Yaskawa INFORM job: SKRZYNIA_5340_0_STOPNI_1OBR.JBI

/JOB
//NAME SKRZYNIA_5340_0_STOPNI_1OBR
///FOLDERNAME 02-SKRZYNIE_JOBS
//POS
///NPOS 610,610,0,47,4,0
///TOOL 0
///POSTYPE PULSE
///PULSE
C00000=1055,-24125,84372,288,19725,204
C00001=1055,-24125,84372,288,19725,204
C00002=0,-15438,65714,0,-68532,0
C00003=25524,-25821,36823,19654,-58495,38520
C00004=23988,-24960,37134,18595,-57837,38812
C00005=22822,-23954,37534,17811,-57199,39017
C00006=22935,-24057,37491,17887,-57262,38997
C00007=20006,-24258,37408,15644,-56932,39751
C00008=24402,-25289,37013,18874,-58060,38740
C00009=22585,-24665,40358,17164,-59622,30036
C00010=23477,-23257,40205,18030,-58646,29630
C00011=22519,-22398,40568,17384,-58125,29795
C00012=22700,-22567,40495,17506,-58225,29764
C00013=19339,-22794,40398,14955,-57865,30607
C00014=24825,-24328,39798,18931,-59350,29401
C00015=32755,-32613,25711,29640,-48730,33694
C00016=25632,-30899,26166,23992,-46203,35378
C00017=24264,-29862,26497,22996,-45413,35639
C00018=24403,-29974,26459,23097,-45496,35612
C00019=20575,-30233,26374,19602,-44891,36810
C00020=26556,-31526,25988,24663,-46720,35206
C00021=30846,-32795,25752,28021,-48338,30427
C00022=24953,-30697,26306,23444,-45946,31743
C00023=23937,-29910,26558,22702,-45353,31936
C00024=24039,-29993,26530,22778,-45414,31916
C00025=20322,-30240,26449,19379,-44834,33080
C00026=25997,-31433,26093,24205,-46535,31545
C00027=26028,-43665,26580,-39946,8682,24640
C00028=27956,-30595,53065,-101898,6609,54413
C00029=26028,-43663,26580,-39944,8677,24639
C00030=38784,-34544,25404,33956,-51320,34445
C00031=29266,-32676,25756,26732,-47889,36488
C00032=25734,-31262,26119,24020,-46377,37252
C00033=24289,-30200,26441,22967,-45549,37525
C00034=24367,-30262,26420,23025,-45594,37511
C00035=20043,-30544,26331,19080,-44922,38860
C00036=26573,-31816,25967,24631,-46839,37095
C00037=27817,-32566,25782,25532,-47502,36865
C00038=25779,-31294,26110,24054,-46400,37243
C00039=24344,-30243,26427,23007,-45578,37515
C00040=24432,-30312,26405,23072,-45630,37498
C00041=20021,-30599,26315,19050,-44944,38872
C00042=26262,-31616,26021,24405,-46667,37153
C00043=27439,-32346,25835,25259,-47302,36935
C00044=25570,-31108,26163,23910,-46262,37277
C00045=24581,-30384,26384,23190,-45695,37464
C00046=24689,-30466,26358,23269,-45758,37444
C00047=20001,-30771,26264,18999,-45026,38899
C00048=26308,-31607,26026,24448,-46671,37139
C00049=27526,-32360,25834,25329,-47326,36914
C00050=24269,-40076,6479,29767,-34177,34232
C00051=22958,-37632,10123,27061,-35370,35326
C00052=22703,-41294,1722,31272,-29953,33282
C00053=19440,-41515,1663,27208,-29122,34832
C00054=25465,-43501,1200,33269,-31905,32752
C00055=87177,-39066,-1236,81808,-72661,19198
C00056=4794,-34097,38974,4189,-31824,-1302
C00057=4794,-34097,38974,4189,13412,-1302
C00058=11237,-37131,38982,-12694,5333,8253
C00059=6591,-33902,35532,5956,-1761,-1932
C00060=10065,-33530,28876,9373,-31104,-3154
C00061=31877,-32319,25770,29025,-48287,33360
C00062=24706,-30765,26196,23236,-45867,35119
C00063=23652,-29939,26460,22464,-45250,35320
C00064=23742,-30013,26436,22530,-45305,35302
C00065=19630,-30281,26348,18756,-44677,36597
C00066=26056,-31710,25928,24219,-46631,34863
C00067=38095,-40136,7813,41252,-44156,24924
C00068=33231,-38681,8176,37792,-41757,25918
C00069=31538,-37640,8473,36716,-40716,26179
C00070=31687,-37737,8444,36811,-40809,26155
C00071=27389,-38154,8322,32773,-39589,27627
C00072=33834,-39023,8084,38175,-42120,25821
C00073=27585,-47842,-289,32095,-40789,28095
C00074=4801,-35772,25187,4593,-28023,-82032
C00075=17634,-23800,39238,9573,-31425,-73339
C00076=17634,-23800,39238,9573,-31425,-73339
C00077=16549,-22464,39800,8390,-30730,-72975
C00078=16684,-22641,39722,8536,-30818,-73021
C00079=16684,-19968,45512,8078,-32771,-72767
C00080=17634,-23800,39238,9573,-31425,-73339
C00081=17837,-21535,44509,9322,-33342,-73155
C00082=17837,-21535,44509,9322,-33342,-73155
C00083=16866,-20378,45014,8305,-32755,-72853
C00084=17032,-20588,44918,8481,-32857,-72905
C00085=17032,-17542,51480,8009,-35060,-72636
C00086=17837,-21535,44509,9322,-33342,-73155
C00087=-20829,-18800,50532,-12466,-37179,-77446
C00088=-19934,-17904,50946,-11618,-36715,-77676
C00089=-20044,-18019,50891,-11723,-36773,-77647
C00090=-20044,-15288,56753,-11218,-38713,-77950
C00091=-20966,-18928,50473,-12596,-37250,-77413
C00092=-20884,-26676,33664,-14451,-31668,-76336
C00093=-20884,-26676,33664,-14451,-31668,-76336
C00094=-19557,-25338,34176,-13080,-30873,-76751
C00095=-19691,-25483,34117,-13220,-30955,-76709
C00096=-19691,-22773,39998,-12506,-32911,-77106
C00097=-20642,-26447,33747,-14206,-31526,-76411
C00098=-33629,-40566,17444,-29603,-33447,-71192
C00099=-33629,-40566,17444,42578,-32312,-84654
C00100=-42160,-31266,16400,42578,-32312,-84654
C00101=-87798,-804,48829,-20188,-26072,-60966
C00102=-76454,-11934,10236,-25964,7954,-64922
C00103=-76448,-11928,10235,-25961,7944,-64914
C00104=-68643,-7759,-23318,-14097,50582,-74897
C00105=-70868,-8793,-8075,-29663,30364,-70765
C00106=-67243,-1968,12282,-49553,26687,-63567
C00107=-68655,-309,14069,-48513,25966,-64203
C00108=-67497,-1678,12591,-49367,26558,-63682
C00109=-71436,-723,2905,-26484,35140,-73726
C00110=-71436,176,6426,-27636,33595,-73066
C00111=-71434,778,8668,-28412,32633,-72624
C00112=-68624,-2689,-85,-28291,36551,-72622
C00113=-99375,3692,5712,40719,48607,-84097
C00114=-94964,4957,10918,40408,44640,-83792
C00115=-93063,6047,12199,39572,43744,-83178
C00116=-94964,4957,10918,40408,44640,-83792
C00117=-94964,5754,13918,41385,43553,-84439
C00118=-94964,4957,10918,40408,44640,-83792
C00119=-90271,-412,-5146,23417,46876,-76529
C00120=-83133,-4088,-8267,6704,41492,-71542
C00121=-83133,-4088,-8267,6704,41492,-71542
C00122=-83133,-4088,-8267,6704,41492,-11598
C00123=-83133,-16026,-8267,6704,41492,-11598
C00124=-83133,-16026,-8267,6704,41492,-11598
C00125=-48225,-19387,30619,3889,32460,-6728
C00126=56943,-39861,25115,1795,-37402,-69601
C00127=29960,-38386,-19607,-115769,-41858,-24264
C00128=65721,-6478,18155,-133323,-22195,3361
C00129=70544,4411,32968,-134868,-18623,4660
C00130=71874,8263,38598,-134556,-17327,4659
C00131=72629,9390,40002,-135279,-16924,5107
C00132=71441,7638,37831,-134139,-17555,4406
C00133=77146,8888,25050,-166574,-32612,18372
C00134=77146,10029,28643,-166204,-31014,18167
C00135=77146,11198,32202,-165803,-29459,17947
C00136=75508,4678,16951,-165715,-35157,17778
C00137=68680,12216,24468,-164340,-40455,-13359
C00138=68362,12845,25743,-164045,-40097,-13561
C00139=68362,13700,28585,-163752,-38808,-13742
C00140=68362,12845,25743,-164045,-40097,-13561
C00141=64993,-1168,28876,-102971,-10760,-49875
C00142=63888,481,30670,-102324,-11438,-50313
C00143=64993,-1168,28876,-102971,-10760,-49875
C00144=4264,-34194,25387,4006,-26954,-29436
C00145=4264,-34194,25387,4006,-26954,-81856
C00146=17634,-23800,39238,9573,-31425,-73339
C00147=17837,-27228,32238,10495,-29236,-73805
C00148=17837,-21535,44509,9322,-33342,-73155
C00149=17548,-20734,45666,8935,-33511,-73021
C00150=-20829,-18800,50532,-12466,-37179,-77446
C00151=-20884,-20901,46110,-12960,-35762,-77182
C00152=-20884,-26676,33664,-14451,-31668,-76336
C00153=-20624,-26699,33167,-14265,-31320,-76369
C00154=-33629,-40566,17444,-29603,-33447,-71192
C00155=-33629,-40566,17444,42578,-32312,-84654
C00156=-42160,-31266,16400,42578,-32312,-84654
C00157=-87798,-804,48829,-20188,-26072,-60966
C00158=-76454,-11934,10236,-25964,7954,-64922
C00159=-76448,-11928,10235,-25961,7944,-64914
C00160=-68643,-7759,-23318,-14097,50582,-74897
C00161=-70868,-8793,-8075,-29663,30364,-70765
C00162=-67243,-1968,12282,-49553,26687,-63567
C00163=-68655,-309,14069,-48513,25966,-64203
C00164=-67497,-1678,12591,-49367,26558,-63682
C00165=-71436,-723,2905,-26484,35140,-73726
C00166=-71436,176,6426,-27636,33595,-73066
C00167=-71434,778,8668,-28412,32633,-72624
C00168=-68624,-2689,-85,-28291,36551,-72622
C00169=-99375,3692,5712,40719,48607,-84097
C00170=-94964,4957,10918,40408,44640,-83792
C00171=-93063,6047,12199,39572,43744,-83178
C00172=-94964,4957,10918,40408,44640,-83792
C00173=-94964,5754,13918,41385,43553,-84439
C00174=-94964,4957,10918,40408,44640,-83792
C00175=-90271,-412,-5146,23417,46876,-76529
C00176=-83133,-4088,-8267,6704,41492,-71542
C00177=-83133,-4088,-8267,6704,41492,-71542
C00178=-83133,-4088,-8267,6704,41492,-11598
C00179=-83133,-16026,-8267,6704,41492,-11598
C00180=-83133,-16026,-8267,6704,41492,-11598
C00181=-48225,-19387,30619,3889,32460,-6728
C00182=56943,-39861,25115,1795,-37402,-69601
C00183=29960,-38386,-19607,-115769,-41858,-24264
C00184=65721,-6478,18155,-133323,-22195,3361
C00185=70544,4411,32968,-134868,-18623,4660
C00186=71874,8263,38598,-134556,-17327,4659
C00187=72629,9390,40002,-135279,-16924,5107
C00188=71441,7638,37831,-134139,-17555,4406
C00189=77146,8888,25050,-166574,-32612,18372
C00190=77146,10029,28643,-166204,-31014,18167
C00191=77146,11198,32202,-165803,-29459,17947
C00192=75508,4678,16951,-165715,-35157,17778
C00193=68680,12216,24468,-164340,-40455,-13359
C00194=68362,12845,25743,-164045,-40097,-13561
C00195=68362,13700,28585,-163752,-38808,-13742
C00196=68362,12845,25743,-164045,-40097,-13561
C00197=64993,-1168,28876,-102971,-10760,-49875
C00198=63888,481,30670,-102324,-11438,-50313
C00199=64993,-1168,28876,-102971,-10760,-49875
C00200=58588,-14653,4620,-120782,-19611,-35794
C00201=29960,-38386,-19607,-115769,-41858,-24264
C00202=56943,-39861,25115,1795,-37402,-69601
C00203=-1002,-39861,25115,1795,-37402,-69601
C00204=-1001,-39858,25114,1795,-37402,0
C00205=6591,-33902,35532,5956,-1761,-1932
C00206=6592,-33900,35531,103508,-35512,-26314
C00207=-99253,-13690,44082,59847,13407,-31313
C00208=-85045,-36869,-4353,28502,-22832,-52282
C00209=-92346,-18713,13565,21110,-22545,-55257
C00210=-85370,-14218,16934,32905,-23649,-60330
C00211=-84150,-13282,17685,34842,-23935,-61163
C00212=-82877,-12536,18624,36445,-24482,-61818
C00213=-84150,-13282,17685,34842,-23935,-61163
C00214=-85467,-11480,19558,33086,-23405,-60436
C00215=-84150,-13282,17685,34842,-23935,-61163
C00216=-85732,-21202,11427,30682,-24763,-59235
C00217=-84559,-15616,15722,33768,-24118,-60665
C00218=-84150,-13282,17685,34842,-23935,-61163
C00219=-83260,-12880,18034,36130,-24218,-61709
C00220=-84150,-13282,17685,34842,-23935,-61163
C00221=-85365,-11775,19006,33430,-23307,-60600
C00222=-84150,-13282,17685,34842,-23935,-61163
C00223=-85786,-16909,14677,31743,-23900,-59790
C00224=-84150,-13282,17685,34842,-23935,-61163
C00225=-83215,-12861,18051,36194,-24233,-61735
C00226=-84150,-13282,17685,34842,-23935,-61163
C00227=-85327,-11825,18959,33476,-23327,-60618
C00228=-84150,-13282,17685,34842,-23935,-61163
C00229=-87841,-18519,13420,28367,-23534,-58339
C00230=-84150,-13282,17685,34842,-23935,-61163
C00231=-83292,-12894,18020,36083,-24208,-61688
C00232=-84150,-13282,17685,34842,-23935,-61163
C00233=-85185,-12008,18799,33646,-23400,-60687
C00234=-84150,-13282,17685,34842,-23935,-61163
C00235=-86371,-18277,13606,30568,-23951,-59265
C00236=-84345,-13370,17612,34554,-23873,-61041
C00237=-83240,-12871,18042,36158,-24225,-61720
C00238=-84345,-13370,17612,34554,-23873,-61041
C00239=-85365,-12110,18711,33368,-23345,-60568
C00240=-84345,-13370,17612,34554,-23873,-61041
C00241=-86191,-19647,12567,30467,-24278,-59187
C00242=-84345,-13372,17610,34552,-23873,-61039
C00243=-83096,-12807,18098,36363,-24268,-61804
C00244=-84345,-13372,17610,34552,-23873,-61039
C00245=-85268,-12232,18600,33480,-23393,-60612
C00246=-84345,-13372,17610,34552,-23873,-61039
C00247=-84814,-16043,15376,33312,-24093,-60464
C00248=-84104,-13265,17702,34906,-23948,-61189
C00249=-82960,-12743,18153,36555,-24313,-61887
C00250=-84104,-13265,17702,34906,-23948,-61189
C00251=-84979,-12194,18635,33901,-23496,-60788
C00252=-84104,-13265,17702,34906,-23948,-61189
C00253=-86610,-16845,14732,30573,-23614,-59301
C00254=-84104,-13265,17702,34906,-23948,-61189
C00255=-82793,-12667,18222,36790,-24370,-61986
C00256=-84104,-13265,17702,34906,-23948,-61189
C00257=-84888,-12305,18537,34004,-23540,-60830
C00258=-84104,-13265,17702,34906,-23948,-61189
C00259=-83806,-19585,12613,33764,-25080,-60559
C00260=-83675,-13072,17868,35530,-24083,-61453
C00261=-82553,-12556,18319,37130,-24451,-62127
C00262=-83675,-13072,17868,35530,-24083,-61453
C00263=-84378,-12223,18610,34735,-23716,-61138
C00264=-83675,-13072,17868,35530,-24083,-61453
C00265=-87149,-17993,13826,29513,-23647,-58830
C00266=-84104,-13265,17702,34906,-23948,-61189
C00267=-82640,-12594,18285,37014,-24425,-62079
C00268=-84104,-13265,17702,34906,-23948,-61189
C00269=-84792,-12429,18430,34119,-23592,-60877
C00270=-84104,-13265,17702,34906,-23948,-61189
C00271=-83583,-9185,30892,23668,-36042,-57025
C00272=-85789,-8328,35795,20592,-37093,-55378
C00273=-85786,-16735,14816,31782,-23869,-59812
C00274=-84103,-13263,17702,34906,-23947,-61191
C00275=-83225,-12865,18046,36177,-24227,-61729
C00276=-84103,-13263,17702,34906,-23947,-61191
C00277=-84774,-12447,18412,34138,-23599,-60886
C00278=-84103,-13263,17702,34906,-23947,-61191
C00279=-86149,-16246,6730,18897,-35239,-57128
C00280=-86244,-15289,7532,18875,-35060,-57127
C00281=-85361,-14893,7870,19824,-35193,-57574
C00282=-86244,-15289,7532,18875,-35060,-57127
C00283=-86889,-14409,8282,18264,-34784,-56850
C00284=-86244,-15289,7532,18875,-35060,-57127
C00285=-90262,-21765,2389,14114,-35574,-54847
C00286=-90262,-21765,2389,28730,-17672,-54847
C00287=-89967,-19086,25635,28730,-17672,-54847
C00288=568,-24029,84339,168,19981,112
C00289=568,-24677,83015,164,20405,113
C00290=101153,-24598,83176,165,20353,113
C00291=101153,-24598,83176,165,20353,113
C00292=89967,-19086,25635,-28730,-17672,54847
C00293=90262,-21765,2389,-28730,-17672,54847
C00294=86932,-18662,4771,-17876,-35519,56628
C00295=86578,-15436,7408,-18515,-35011,56957
C00296=85428,-14922,7844,-19753,-35183,57541
C00297=84405,-14447,8250,-20842,-35348,58054
C00298=85428,-14922,7844,-19753,-35183,57541
C00299=86134,-13973,8661,-19091,-34881,57237
C00300=85428,-14922,7844,-19753,-35183,57541
C00301=85786,-16735,14816,-31782,-23869,59812
C00302=83514,-12996,17929,-35760,-24132,61552
C00303=82296,-12429,18424,-37488,-24534,62281
C00304=83514,-12996,17929,-35760,-24132,61552
C00305=84266,-12085,18725,-34910,-23738,61214
C00306=83514,-12996,17929,-35760,-24132,61552
C00307=87323,-6914,39851,-18853,-38149,44508
C00308=83118,-12818,18089,-36330,-24263,61791
C00309=81969,-12276,18566,-37944,-24648,62472
C00310=83118,-12818,18089,-36330,-24263,61791
C00311=83927,-11846,18941,-35423,-23842,61433
C00312=83118,-12818,18089,-36330,-24263,61791
C00313=83806,-19585,12613,-33764,-25080,60559
C00314=83148,-12832,18077,-36287,-24254,61773
C00315=81889,-12236,18598,-38058,-24676,62520
C00316=83148,-12832,18077,-36287,-24254,61773
C00317=83900,-11930,18867,-35446,-23862,61440
C00318=83148,-12832,18077,-36287,-24254,61773
C00319=86610,-16845,14732,-30573,-23614,59301
C00320=82493,-13239,17725,-37070,-24559,62089
C00321=81442,-12739,18159,-38529,-24915,62703
C00322=82493,-13239,17725,-37070,-24559,62089
C00323=83435,-12133,18689,-36040,-24063,61682
C00324=82493,-13239,17725,-37070,-24559,62089
C00325=84814,-16043,15376,-33312,-24093,60464
C00326=82555,-13613,17404,-36910,-24580,62015
C00327=81369,-13053,17885,-38558,-24979,62709
C00328=82555,-13613,17404,-36910,-24580,62015
C00329=83568,-12431,18429,-35805,-24046,61580
C00330=82555,-13613,17404,-36910,-24580,62015
C00331=86191,-19647,12567,-30467,-24278,59187
C00332=82500,-13648,17375,-36975,-24607,62039
C00333=81594,-13224,17740,-38236,-24911,62571
C00334=82500,-13648,17375,-36975,-24607,62039
C00335=83449,-12543,18332,-35941,-24104,61633
C00336=82500,-13648,17375,-36975,-24607,62039
C00337=86371,-18277,13606,-30568,-23951,59265
C00338=82904,-13790,17251,-36416,-24470,61808
C00339=81796,-13275,17692,-37971,-24838,62464
C00340=82904,-13790,17251,-36416,-24470,61808
C00341=83696,-12867,18046,-35547,-24051,61466
C00342=82904,-13790,17251,-36416,-24470,61808
C00343=87841,-18519,13420,-28367,-23534,58339
C00344=82748,-13879,17174,-36603,-24542,61883
C00345=81789,-13434,17554,-37946,-24861,62449
C00346=82748,-13879,17174,-36603,-24542,61883
C00347=83603,-12888,18026,-35668,-24086,61514
C00348=82748,-13879,17174,-36603,-24542,61883
C00349=85786,-16909,14677,-31743,-23900,59790
C00350=82339,-14116,16972,-37087,-24733,62079
C00351=81557,-13752,17280,-38171,-24994,62536
C00352=82339,-14116,16972,-37087,-24733,62079
C00353=83390,-12909,18006,-35951,-24172,61633
C00354=82339,-14116,16972,-37087,-24733,62079
C00355=85732,-21202,11427,-30682,-24763,59235
C00356=82398,-14365,16763,-36952,-24745,62014
C00357=81340,-13876,17176,-38416,-25096,62632
C00358=82398,-14365,16763,-36952,-24745,62014
C00359=83629,-12951,17972,-35620,-24090,61491
C00360=82398,-14365,16763,-36952,-24745,62014
C00361=92346,-18713,13565,-21110,-22545,55257
C00362=82794,-13980,17083,-36511,-24538,61844
C00363=81697,-13472,17516,-38043,-24902,62488
C00364=82794,-13980,17083,-36511,-24538,61844
C00365=83767,-12847,18056,-35444,-24023,61424
C00366=82794,-13980,17083,-36511,-24538,61844
C00367=85045,-36869,-4353,-28502,-22832,52282
C00368=69856,-53931,-13446,-33557,-28911,29591
C00369=73943,-28815,39553,-16801,-45089,19004
C00370=0,-24029,84339,0,19981,0
C00371=0,-24029,84339,0,19981,0
C00372=0,-52280,40443,0,6876,0
C00373=63961,-36661,14391,66570,-58199,13439
C00374=50233,-31965,16595,55443,-54435,15843
C00375=47147,-32819,12541,55607,-51124,17230
C00376=46896,-37872,871,62973,-46008,11193
C00377=54160,-39955,137,66075,-50361,10746
C00378=0,-52280,40443,0,6876,0
C00379=0,-52280,40443,1,6876,0
C00380=42978,-45587,7631,48214,-41849,18034
C00381=34615,-32719,24207,35617,-45539,22507
C00382=46734,-24688,30880,50025,-55713,21863
C00383=45059,-39151,-3508,69830,-41334,11649
C00384=32474,-45233,-13338,65386,-28486,22104
C00385=59828,-44646,-5405,72855,-48572,12139
C00386=0,-38761,66314,0,-763,0
C00387=0,-44757,54667,0,2744,0
C00388=40382,-38226,12225,48505,-40693,16039
C00389=55481,-27484,23768,62968,-54833,11978
C00390=49931,-26522,24223,59987,-51967,12537
C00391=49591,-31309,12277,55066,-55958,13102
C00392=55330,-33748,11238,57660,-59334,12681
C00393=78664,-24436,10378,82837,-79111,12029
C00394=75189,-23065,11287,81851,-76948,11927
C00395=75189,-45249,11287,81851,-38847,11927
C00396=29880,-45249,11287,43145,-11324,11927
C00397=0,-24029,84339,0,19981,0
C00398=0,-24026,84338,1,19977,2
C00399=4264,-34194,25387,4006,-26954,-29436
C00400=4264,-34194,25387,4006,-26954,-81856
C00401=-21478,-27798,32214,-15234,-31599,-76056
C00402=-19679,-23059,39354,-12567,-32689,-77067
C00403=16724,-20576,44291,8212,-32395,-72836
C00404=21329,-26386,39716,13285,-34016,-74401
C00405=-23778,-26243,38799,-16502,-35132,-75964
C00406=-20075,-15782,55752,-11329,-38404,-77896
C00407=16874,-17447,51356,7863,-34895,-72604
C00408=18580,-28601,30698,11472,-29284,-74138
C00409=6126,-41331,18955,6697,-26557,-30383
C00410=1,-24024,84337,2,19973,1
C00411=-64243,-26178,31107,-39513,40312,-5844
C00412=-72148,3973,56008,-35470,42045,-10522
C00413=-72090,16396,76301,-42067,35650,-6519
C00414=-69388,15725,61378,-31740,35177,-8719
C00415=-69127,27099,75569,-32744,34250,-8088
C00416=-67573,2495,11285,-21767,57629,-15193
C00417=-77819,19629,29798,-10454,63174,-20704
C00418=-72990,23583,14304,-10735,77209,-20379
C00419=-74593,38003,46707,-11043,65751,-19814
C00420=-73236,38943,48295,-11400,65557,-19316
C00421=-73329,42107,51779,-6346,67443,-19636
C00422=-87142,34654,46174,17622,63862,-25393
C00423=-87240,36727,48611,18897,66604,-25032
C00424=-99033,21517,12213,24947,79702,-26203
C00425=-91500,-14196,-34781,24472,81625,-22832
C00426=-100472,-45007,-27818,8167,67201,-29302
C00427=0,-36642,16905,0,48372,0
C00428=66009,-61997,-62105,21406,63483,18379
C00429=97242,-23579,-39442,10179,68876,30321
C00430=73684,-7073,-17511,24638,68131,29022
C00431=59136,7235,6676,33270,66602,27507
C00432=54816,14937,6234,39741,69494,31070
C00433=54365,20668,19279,41017,66202,29418
C00434=64503,4223,2857,29650,48528,26647
C00435=75622,3202,-3149,3890,49494,34281
C00436=88036,13177,2413,-18568,66573,35876
C00437=90462,21593,10123,-22613,76266,34479
C00438=92450,29224,20002,-25750,81642,33727
C00439=94949,8131,-12163,-20291,74229,36861
C00440=94949,8084,-13484,-20215,75047,36712
C00441=70412,-34016,-52305,-11724,65624,29757
C00442=18580,-28601,30698,11472,-29284,-74138
C00443=-23778,-26243,38799,-16502,-35132,-75964
C00444=18580,-28601,30698,11472,-29284,-74138
C00445=4264,-34194,25387,4006,-26954,-81856
C00446=4264,-34194,25387,4006,-26954,-29436
C00447=1,-24024,84337,2,19973,1
C00448=-64243,-26178,31107,-39513,40312,-5844
C00449=-72148,3973,56008,-35470,42045,-10522
C00450=-72090,16396,76301,-42067,35650,-6519
C00451=-69388,15725,61378,-31740,35177,-8719
C00452=-69127,27099,75569,-32744,34250,-8088
C00453=-67573,2495,11285,-21767,57629,-15193
C00454=-77819,19629,29798,-10454,63174,-20704
C00455=-72990,23583,14304,-10735,77209,-20379
C00456=-74593,38003,46707,-11043,65751,-19814
C00457=-73236,38943,48295,-11400,65557,-19316
C00458=-73329,42107,51779,-6346,67443,-19636
C00459=-87142,34654,46174,17622,63862,-25393
C00460=-87240,36727,48611,18897,66604,-25032
C00461=-99033,21517,12213,24947,79702,-26203
C00462=-91500,-14196,-34781,24472,81625,-22832
C00463=-100472,-45007,-27818,8167,67201,-29302
C00464=0,-36642,16905,0,48372,0
C00465=66009,-61997,-62105,21406,63483,18379
C00466=97242,-23579,-39442,10179,68876,30321
C00467=73684,-7073,-17511,24638,68131,29022
C00468=59136,7235,6676,33270,66602,27507
C00469=54816,14937,6234,39741,69494,31070
C00470=54365,20668,19279,41017,66202,29418
C00471=64503,4223,2857,29650,48528,26647
C00472=75622,3202,-3149,3890,49494,34281
C00473=88036,13177,2413,-18568,66573,35876
C00474=90462,21593,10123,-22613,76266,34479
C00475=92450,29224,20002,-25750,81642,33727
C00476=94949,8131,-12163,-20291,74229,36861
C00477=94949,8084,-13484,-20215,75047,36712
C00478=70412,-34016,-52305,-11724,65624,29757
C00479=44268,-30306,-1568,-7370,48673,18708
C00480=1,-24024,84337,2,19973,1
C00481=1,-24024,84337,2,19973,1
C00482=3796,-57671,22373,2336,-25309,-753
C00483=52632,-34554,16626,51161,-63050,5622
C00484=59461,-32779,9832,66317,-58406,17312
C00485=52745,-27759,19165,60340,-56543,14824
C00486=51596,-17381,41670,51728,-64721,19335
C00487=62932,-33588,12189,66848,-61063,18031
C00488=1,-24024,84337,2,19973,1
C00489=1,-24024,84337,2,19973,1
C00490=57188,-41777,19973,48132,-58706,4905
C00491=55566,-48748,-16991,79805,-45048,-6941
C00492=49908,-48716,-25784,90749,-41340,-3650
C00493=44060,-47282,-25482,90760,-37623,-4446
C00494=43373,-46910,-25348,90885,-37191,-4606
C00495=55479,-50244,-26473,91085,-44870,-3042
C00496=12119,-24859,71505,13236,4440,2633
C00497=-91085,-34291,10385,1908,-24348,-42097
C00498=-86191,-19647,12567,30467,-24278,-59187
C00499=-99148,-11667,19101,-13975,-20192,-40187
C00500=-98206,-11518,19604,-10142,-20308,-41629
C00501=-99474,-20389,12397,-11593,-22150,-41069
C00502=0,-52280,40443,0,6876,0
C00503=85348,-24204,23536,-13963,-15515,44275
C00504=84670,-17015,14597,-33277,-24304,60423
C00505=96971,-12584,18294,8365,-19955,42614
C00506=97182,-12918,18001,8747,-20027,42449
C00507=96230,-24528,9149,6144,-22576,43630
C00508=0,-52280,40443,0,6876,0
C00509=0,-52280,40443,0,6876,0
C00510=-90140,-60305,18108,-2708,1721,-7625
C00511=-95594,-27428,6866,-4663,-19832,-42154
C00512=-99356,-13410,18355,-15385,-17730,-37479
C00513=-99405,-10878,20508,-15853,-17333,-37255
C00514=-99132,-10804,20575,-15274,-17279,-37502
C00515=-99132,-3482,39129,-10940,-24351,-39674
C00516=-98851,-3328,38974,-10588,-24101,-39807
C00517=-100183,-18601,14070,-16273,-18800,-37146
C00518=-90140,-60305,18108,-2708,1721,-7625
C00519=0,-52280,40443,0,6876,0
C00520=84259,-57935,27522,-3761,3673,6310
C00521=86507,-39672,4297,-27618,-16640,46340
C00522=70477,-27878,7073,-45786,-32339,64941
C00523=84043,-16293,15174,-34312,-24409,60872
C00524=94507,-13191,17794,-563,-19874,46473
C00525=99154,-17369,4403,32227,-9753,28926
C00526=99154,-17369,4403,32227,-9753,28926
C00527=98946,-17182,4556,31649,-9649,29182
C00528=100388,-17987,13832,15751,-21517,39479
C00529=86507,-39672,4297,-27618,-16640,46340
C00530=84259,-57935,27522,-3761,3673,6310
C00531=0,-52280,40443,0,6876,0
C00532=0,-27933,77061,0,20812,0
C00533=0,-27933,77061,0,20812,0
C00534=0,-52280,40443,0,6876,0
C00535=-91970,-60791,14435,-3343,512,-9412
C00536=-99196,-15868,16098,-13748,-19297,-38710
C00537=-99196,-15868,16098,-13748,-19297,-38710
C00538=-99196,-15868,16098,-13748,-19297,-38710
C00539=-85815,-11758,19597,31748,-21097,-58265
C00540=-87383,-11883,19487,26986,-20206,-56250
C00541=-99562,-16264,15781,-14410,-19427,-38431
C00542=-99196,-15868,16098,-13748,-19297,-38710
C00543=-91970,-60791,14435,-3343,512,-9412
C00544=0,-52280,40443,0,6876,0
C00545=91083,-60784,14823,-9043,-825,15173
C00546=83869,-19403,12921,-33769,-24740,60260
C00547=83869,-19403,12921,-33769,-24740,60260
C00548=83420,-14897,16486,-35538,-24144,61113
C00549=90535,-11845,19652,-14037,-20800,51549
C00550=90317,-11662,19878,-14346,-20882,51648
C00551=95871,-14889,15992,4901,-19605,43825
C00552=83869,-19403,12921,-33769,-24740,60260
C00553=91083,-60784,14823,-9043,-825,15173
C00554=0,-52280,40443,0,6876,0
C00555=-91526,-60598,16699,7584,176,-13289
C00556=-94392,-6553,48683,5805,-47321,-49764
C00557=-88951,-345,54953,10686,-47392,-51569
C00558=-88172,5833,62122,11322,-47753,-51785
C00559=-90949,-14015,9500,8834,-34399,-51934
C00560=-84917,-15593,15742,33275,-23984,-60461
C00561=-81669,-15982,15425,37506,-25258,-62202
C00562=-79867,-25377,9541,37586,-25936,-59971
C00563=-91415,-60262,16631,7870,-73,-13734
C00564=24,-24029,84339,7,19981,5
C00565=160,-24029,84339,47,19981,32
C00566=99096,-24029,84339,47,19981,32
C00567=99096,-24029,84339,47,19981,32
C00568=89967,-19086,25635,-28730,-17672,54847
C00569=85786,-16735,14816,-31782,-23869,59812
C00570=83492,-14473,16674,-35480,-24338,61406
C00571=82709,-11470,19305,-37370,-24374,62232
C00572=85293,-13629,8874,-19696,-34851,57583
C00573=85505,-16299,6686,-19564,-35388,57437
C00574=89967,-19086,25635,-28730,-17672,54847
C00575=568,-24029,84339,168,19981,112
C00576=568,-24029,84339,168,19981,112
C00577=-91970,-60791,14435,-3343,512,-9412
C00578=-86948,-23217,10819,28314,-23349,-56438
C00579=-85895,-16522,15767,31843,-22281,-58087
C00580=-93643,1708,52973,2937,-38210,-34777
C00581=-93409,-737,47229,3345,-36106,-34967
C00582=-86145,-24679,9854,29028,-23971,-56682
C00583=-100471,-58311,4157,14142,-4822,-27614
C00584=-68517,-58311,4157,14142,-4822,-27614
C00585=0,-52280,40443,0,6876,0
C00586=91083,-60784,14823,-9043,-825,15173
C00587=83869,-19403,12921,-33769,-24740,60260
C00588=82620,-18743,14708,-32942,-26226,58979
C00589=83315,-11405,20766,-33572,-24860,59408
C00590=83326,-11144,20997,-33599,-24827,59423
C00591=84798,-22668,11879,-29033,-26372,57255
C00592=91083,-60784,14823,-9043,-825,15173
C00593=0,-52280,40443,0,6876,0
C00594=-6369,-39206,65423,-4801,-482,2563
C00595=-97287,-29142,12714,-8673,-22288,-37832
C00596=-86191,-19647,12567,30467,-24278,-59187
C00597=-85671,-16302,15857,30808,-24404,-58999
C00598=-99965,-10410,22406,-14600,-22538,-38834
C00599=-95758,-10871,21797,-1120,-21702,-44724
C00600=-87910,-17792,15835,25414,-24996,-56048
C00601=-97287,-29142,12714,-8673,-22288,-37832
C00602=0,-52280,40443,0,6876,0
C00603=92301,-25634,22749,2368,-15645,37646
C00604=83738,-18329,13570,-34202,-24868,60772
C00605=90096,-13099,18146,-15422,-20883,52700
C00606=93330,-13245,17928,-4627,-20146,48105
C00607=80226,-20465,12178,-39626,-27411,62762
C00608=92301,-25634,22749,2368,-15645,37646
C00609=0,-52280,40443,0,6876,0
BC00000=413138
BC00001=413138
BC00002=413138
BC00003=413134
BC00004=413134
BC00005=413134
BC00006=413134
BC00007=413134
BC00008=413134
BC00009=474623
BC00010=474628
BC00011=474628
BC00012=474628
BC00013=474628
BC00014=474628
BC00015=522849
BC00016=522849
BC00017=522849
BC00018=522849
BC00019=522849
BC00020=522849
BC00021=586045
BC00022=586045
BC00023=586045
BC00024=586045
BC00025=586045
BC00026=586045
BC00027=479622
BC00028=618860
BC00029=673957
BC00030=663090
BC00031=663090
BC00032=663090
BC00033=663090
BC00034=663090
BC00035=663090
BC00036=663090
BC00037=708270
BC00038=708270
BC00039=708270
BC00040=708270
BC00041=708270
BC00042=708270
BC00043=770184
BC00044=770184
BC00045=770184
BC00046=770184
BC00047=770184
BC00048=770184
BC00049=823730
BC00050=829967
BC00051=829969
BC00052=829970
BC00053=829970
BC00054=829970
BC00055=838761
BC00056=740349
BC00057=687700
BC00058=771943
BC00059=861898
BC00060=900223
BC00061=904141
BC00062=901229
BC00063=901229
BC00064=901229
BC00065=901229
BC00066=901229
BC00067=949836
BC00068=949836
BC00069=949836
BC00070=949836
BC00071=949836
BC00072=965197
BC00073=995919
BC00074=941874
BC00075=957235
BC00076=957235
BC00077=957235
BC00078=957235
BC00079=957235
BC00080=957235
BC00081=961681
BC00082=961681
BC00083=961681
BC00084=961681
BC00085=961681
BC00086=961681
BC00087=961681
BC00088=961681
BC00089=961681
BC00090=961681
BC00091=961681
BC00092=961681
BC00093=961681
BC00094=961681
BC00095=961681
BC00096=961681
BC00097=961681
BC00098=961681
BC00099=961681
BC00100=961681
BC00101=961681
BC00102=961681
BC00103=979433
BC00104=990519
BC00105=1007223
BC00106=1007223
BC00107=1007223
BC00108=1007223
BC00109=1007223
BC00110=1007223
BC00111=1007224
BC00112=1007224
BC00113=1007224
BC00114=1007224
BC00115=1007224
BC00116=1007224
BC00117=1007224
BC00118=1007224
BC00119=997601
BC00120=982967
BC00121=957702
BC00122=957702
BC00123=957702
BC00124=924520
BC00125=890087
BC00126=961681
BC00127=961681
BC00128=961681
BC00129=977895
BC00130=983056
BC00131=983056
BC00132=983056
BC00133=983056
BC00134=983056
BC00135=983056
BC00136=983056
BC00137=983056
BC00138=983056
BC00139=983056
BC00140=983056
BC00141=983056
BC00142=983056
BC00143=983056
BC00144=926513
BC00145=957235
BC00146=941874
BC00147=941874
BC00148=946320
BC00149=946320
BC00150=946320
BC00151=946320
BC00152=946320
BC00153=946320
BC00154=946320
BC00155=946320
BC00156=946320
BC00157=946320
BC00158=946320
BC00159=964072
BC00160=975158
BC00161=991862
BC00162=991862
BC00163=991862
BC00164=991862
BC00165=991862
BC00166=991862
BC00167=991863
BC00168=991863
BC00169=991863
BC00170=991863
BC00171=991863
BC00172=991863
BC00173=991863
BC00174=991863
BC00175=982240
BC00176=967606
BC00177=942341
BC00178=942341
BC00179=942341
BC00180=909159
BC00181=874726
BC00182=946320
BC00183=946320
BC00184=946320
BC00185=962534
BC00186=967695
BC00187=967695
BC00188=967695
BC00189=967695
BC00190=967695
BC00191=967695
BC00192=967695
BC00193=967695
BC00194=967695
BC00195=967695
BC00196=967695
BC00197=967695
BC00198=967695
BC00199=967695
BC00200=962182
BC00201=946320
BC00202=915598
BC00203=915598
BC00204=930961
BC00205=861898
BC00206=861901
BC00207=861901
BC00208=931504
BC00209=963634
BC00210=963631
BC00211=963631
BC00212=963631
BC00213=963631
BC00214=963631
BC00215=963631
BC00216=902188
BC00217=902188
BC00218=902188
BC00219=902188
BC00220=902188
BC00221=902188
BC00222=902188
BC00223=840744
BC00224=840744
BC00225=840744
BC00226=840744
BC00227=840744
BC00228=840744
BC00229=779300
BC00230=779300
BC00231=779300
BC00232=779300
BC00233=779300
BC00234=779300
BC00235=717855
BC00236=717855
BC00237=717855
BC00238=717855
BC00239=717855
BC00240=717855
BC00241=656405
BC00242=656405
BC00243=656405
BC00244=656405
BC00245=656405
BC00246=656405
BC00247=594961
BC00248=594961
BC00249=594961
BC00250=594961
BC00251=594961
BC00252=594961
BC00253=533517
BC00254=533517
BC00255=533517
BC00256=533517
BC00257=533517
BC00258=533517
BC00259=472073
BC00260=472073
BC00261=472073
BC00262=472073
BC00263=472073
BC00264=472073
BC00265=410629
BC00266=410629
BC00267=410629
BC00268=410629
BC00269=410629
BC00270=410629
BC00271=410629
BC00272=349186
BC00273=349186
BC00274=349186
BC00275=349186
BC00276=349186
BC00277=349186
BC00278=349186
BC00279=336469
BC00280=336469
BC00281=336469
BC00282=336469
BC00283=336469
BC00284=336469
BC00285=336469
BC00286=336469
BC00287=336469
BC00288=336469
BC00289=511557
BC00290=512005
BC00291=363797
BC00292=336469
BC00293=336469
BC00294=337415
BC00295=337415
BC00296=337415
BC00297=337415
BC00298=337415
BC00299=337415
BC00300=337415
BC00301=349186
BC00302=350137
BC00303=350137
BC00304=350137
BC00305=350137
BC00306=350137
BC00307=410629
BC00308=411580
BC00309=411580
BC00310=411580
BC00311=411580
BC00312=411580
BC00313=472073
BC00314=473025
BC00315=473025
BC00316=473025
BC00317=473025
BC00318=473025
BC00319=533517
BC00320=534468
BC00321=534468
BC00322=534468
BC00323=534468
BC00324=534468
BC00325=594961
BC00326=594961
BC00327=594961
BC00328=594961
BC00329=594961
BC00330=594961
BC00331=656405
BC00332=657350
BC00333=657350
BC00334=657350
BC00335=657350
BC00336=657350
BC00337=717855
BC00338=718799
BC00339=718799
BC00340=718799
BC00341=718799
BC00342=718799
BC00343=779300
BC00344=780245
BC00345=780245
BC00346=780245
BC00347=780245
BC00348=780245
BC00349=840744
BC00350=841691
BC00351=841691
BC00352=841691
BC00353=841691
BC00354=841691
BC00355=902188
BC00356=903136
BC00357=903136
BC00358=903136
BC00359=903136
BC00360=903136
BC00361=963634
BC00362=963633
BC00363=963633
BC00364=963633
BC00365=963633
BC00366=963633
BC00367=931504
BC00368=861901
BC00369=861901
BC00370=769966
BC00371=769966
BC00372=716865
BC00373=668657
BC00374=668657
BC00375=668657
BC00376=717171
BC00377=717171
BC00378=716865
BC00379=800897
BC00380=908887
BC00381=899019
BC00382=895607
BC00383=945882
BC00384=955598
BC00385=945882
BC00386=840120
BC00387=538973
BC00388=485226
BC00389=456696
BC00390=456696
BC00391=417276
BC00392=417276
BC00393=493986
BC00394=514306
BC00395=514306
BC00396=514306
BC00397=493986
BC00398=797003
BC00399=895791
BC00400=911152
BC00401=961681
BC00402=961681
BC00403=957234
BC00404=951468
BC00405=946979
BC00406=961681
BC00407=961681
BC00408=960909
BC00409=964501
BC00410=812362
BC00411=827724
BC00412=827724
BC00413=884434
BC00414=904320
BC00415=929259
BC00416=961191
BC00417=961191
BC00418=988700
BC00419=988700
BC00420=988700
BC00421=988701
BC00422=988701
BC00423=988702
BC00424=988702
BC00425=988702
BC00426=903360
BC00427=861958
BC00428=945498
BC00429=984618
BC00430=984619
BC00431=984619
BC00432=1014866
BC00433=1014866
BC00434=1014866
BC00435=1014866
BC00436=1014866
BC00437=1014869
BC00438=1014869
BC00439=1014869
BC00440=988463
BC00441=988463
BC00442=895791
BC00443=900237
BC00444=895791
BC00445=895791
BC00446=895791
BC00447=797001
BC00448=812363
BC00449=812363
BC00450=869073
BC00451=888959
BC00452=913898
BC00453=945830
BC00454=945830
BC00455=973339
BC00456=973339
BC00457=973339
BC00458=973340
BC00459=973340
BC00460=973341
BC00461=973341
BC00462=973341
BC00463=887999
BC00464=846597
BC00465=930137
BC00466=969257
BC00467=969258
BC00468=969258
BC00469=999505
BC00470=999505
BC00471=999505
BC00472=999505
BC00473=999505
BC00474=999508
BC00475=999508
BC00476=999508
BC00477=973102
BC00478=973102
BC00479=904289
BC00480=812362
BC00481=476651
BC00482=522561
BC00483=566531
BC00484=593948
BC00485=593948
BC00486=529848
BC00487=529848
BC00488=461290
BC00489=663315
BC00490=778314
BC00491=778312
BC00492=778312
BC00493=778312
BC00494=838222
BC00495=838222
BC00496=566410
BC00497=679663
BC00498=656405
BC00499=656405
BC00500=717855
BC00501=717855
BC00502=717855
BC00503=662303
BC00504=657350
BC00505=657350
BC00506=718803
BC00507=718803
BC00508=717855
BC00509=792672
BC00510=792672
BC00511=896850
BC00512=895720
BC00513=895720
BC00514=957178
BC00515=957178
BC00516=978461
BC00517=957178
BC00518=792672
BC00519=792672
BC00520=792672
BC00521=887446
BC00522=903126
BC00523=903126
BC00524=903126
BC00525=964577
BC00526=976097
BC00527=993812
BC00528=964577
BC00529=887446
BC00530=792672
BC00531=792672
BC00532=700249
BC00533=546214
BC00534=546214
BC00535=546211
BC00536=546211
BC00537=406776
BC00538=406776
BC00539=406778
BC00540=468200
BC00541=468200
BC00542=546211
BC00543=546211
BC00544=546214
BC00545=546214
BC00546=507604
BC00547=410782
BC00548=410782
BC00549=410782
BC00550=472720
BC00551=472720
BC00552=507604
BC00553=546214
BC00554=546214
BC00555=516757
BC00556=383716
BC00557=349186
BC00558=349186
BC00559=336469
BC00560=349186
BC00561=410629
BC00562=416512
BC00563=515801
BC00564=520018
BC00565=474013
BC00566=474013
BC00567=403108
BC00568=336469
BC00569=349186
BC00570=349186
BC00571=349186
BC00572=337415
BC00573=337415
BC00574=336469
BC00575=336469
BC00576=428401
BC00577=546211
BC00578=591088
BC00579=591088
BC00580=591088
BC00581=531116
BC00582=529640
BC00583=529640
BC00584=529640
BC00585=529640
BC00586=546214
BC00587=589919
BC00588=595627
BC00589=595627
BC00590=534177
BC00591=534177
BC00592=546214
BC00593=529640
BC00594=651195
BC00595=765890
BC00596=777968
BC00597=778453
BC00598=779252
BC00599=840748
BC00600=840748
BC00601=765890
BC00602=717855
BC00603=741100
BC00604=780224
BC00605=780222
BC00606=841743
BC00607=841743
BC00608=741100
BC00609=717855
///POSTYPE BASE
///RECTAN
///RCONF 1,0,0,0,0,0,0,0,0,0,0,0,0,0,0,0,0,0,0,0,0,0,0,0
P00006=0.000,0.000,0.000,0.0000,0.0000,0.0000
///RCONF 0,0,0,0,0,0,0,0,0,0,0,0,0,0,0,0,0,0,0,0,0,0,0,0
P00021=6.550,-0.003,-5.735,0.0000,0.0000,0.0000
P00022=5.943,-0.018,-6.388,0.0000,0.0000,0.0000
P00023=7.025,-0.019,-7.168,0.0000,0.0000,0.0000
P00024=5.926,-0.047,-4.777,0.0000,0.0000,0.0000
///RCONF 1,0,0,0,0,0,0,0,0,0,0,0,0,0,0,0,0,0,0,0,0,0,0,0
P00100=-0.081,2.558,4.482,0.0000,0.0000,0.0000
P00101=0.030,-2.286,2.993,0.0000,0.0000,0.0000
P00102=-0.005,-1.108,1.644,0.0000,0.0000,0.0000
P00103=-0.094,-3.400,4.200,0.0000,0.0000,0.0000
P00104=0.043,-2.127,5.826,0.0000,0.0000,0.0000
P00105=-0.043,0.662,5.286,0.0000,0.0000,0.0000
P00106=-0.018,-2.519,0.237,0.0000,0.0000,0.0000
P00107=-0.008,-4.537,-4.500,0.0000,0.0000,0.0000
P00108=0.014,-3.040,2.637,0.0000,0.0000,0.0000
P00109=0.017,-3.622,2.341,0.0000,0.0000,0.0000
P00110=7346.140,158.997,-946.107,-0.1876,37.7131,-155.1643
P00111=7345.905,-141.160,-945.062,8.1413,34.2244,-174.1788
P00112=7393.287,158.977,-939.640,-0.1938,37.7128,-155.1905
P00113=7393.259,-141.170,-939.228,8.1507,34.2195,-174.1496
///RCONF 0,0,0,0,0,0,0,0,0,0,0,0,0,0,0,0,0,0,0,0,0,0,0,0
P00280=-0.761,-1.221,0.004,0.0000,0.0000,0.0000
///RCONF 1,0,0,0,0,0,0,0,0,0,0,0,0,0,0,0,0,0,0,0,0,0,0,0
P00281=-0.866,-3.587,-0.008,0.0000,0.0000,0.0000
///RCONF 0,0,0,0,1,0,0,0,0,0,0,0,0,0,0,0,0,0,0,0,0,0,0,0
P00290=-0.023,-0.050,5.560,0.0000,0.0000,0.0000
///RCONF 1,0,0,0,0,0,0,0,0,0,0,0,0,0,0,0,0,0,0,0,0,0,0,0
P00291=0.002,-0.893,4.526,0.0000,0.0000,0.0000
P00300=-0.036,-1.505,2.318,0.0000,0.0000,0.0000
P00301=0.046,-2.112,7.779,0.0000,0.0000,0.0000
P00302=-0.180,-2.409,6.326,0.0000,0.0000,0.0000
///RCONF 0,0,0,0,0,0,0,0,0,0,0,0,0,0,0,0,0,0,0,0,0,0,0,0
P00303=-0.004,-1.437,-4.584,0.0000,0.0000,0.0000
P00304=0.028,-1.666,-4.234,0.0000,0.0000,0.0000
P00305=-0.003,-1.920,-3.501,0.0000,0.0000,0.0000
P00306=0.015,-2.252,-3.054,0.0000,0.0000,0.0000
P00307=0.019,-2.151,-5.077,0.0000,0.0000,0.0000
P00308=-0.003,-2.092,-4.888,0.0000,0.0000,0.0000
P00309=-0.040,-2.205,-4.992,0.0000,0.0000,0.0000
P00310=-0.006,-2.490,-5.925,0.0000,0.0000,0.0000
P00311=-0.007,-2.079,-5.307,0.0000,0.0000,0.0000
P00350=11.519,-0.008,1.149,0.0000,0.0000,0.0000
P00351=13.563,-0.027,-0.653,0.0000,0.0000,0.0000
P00352=13.252,-0.027,-0.827,0.0000,0.0000,0.0000
P00353=10.971,-0.082,0.776,0.0000,0.0000,0.0000
P00354=-0.024,2.508,-1.824,0.0000,0.0000,0.0000
P00355=-0.001,2.528,-1.131,0.0000,0.0000,0.0000
P00356=-0.034,2.921,-0.262,0.0000,0.0000,0.0000
P00357=0.003,3.386,-0.091,0.0000,0.0000,0.0000
P00358=0.014,3.037,-0.020,0.0000,0.0000,0.0000
P00359=-0.005,2.731,0.912,0.0000,0.0000,0.0000
P00360=-0.011,3.412,0.438,0.0000,0.0000,0.0000
P00361=0.018,3.050,1.253,0.0000,0.0000,0.0000
BP00110=5931.608
BP00111=5960.552
BP00112=5960.545
BP00113=5960.552
//INST
///DATE 2024/08/01 13:27
///ATTR SC,RW
///GROUP1 RB1,BS1
NOP
CALL JOB:MOVE_INTO_TUNNEL
MOVJ C00000 BC00000 VJ=30.00
'------------------------
'------------------------
'SPOINA SRODEK DOL
'------------------------
'------------------------
'POMIAR DO WYJ!! PRZEROBIC NA STD
MOVJ C00001 BC00001 VJ=40.00
MOVJ C00002 BC00002 VJ=40.00
'W3P
MOVJ C00003 BC00003 VJ=20.00 PL=0
MOVL C00004 BC00004 V=166.7 PL=0
REFP 3 C00005 BC00005
CALL JOB:SEARCH-R1
SET P0100 P0006
SFTON P0100
MOVL C00006 BC00006 V=66.7 PL=0
REFP 3 C00007 BC00007
CALL JOB:SEARCH-R1
SET P0100 P0006
SFTON P0100
MOVL C00008 BC00008 V=333.3 PL=0
SFTOF
'W3L
MOVL C00009 BC00009 V=666.7
MOVL C00010 BC00010 V=166.7 PL=0
REFP 3 C00011 BC00011
CALL JOB:SEARCH-R1
SET P0101 P0006
SFTON P0101
MOVL C00012 BC00012 V=166.7 PL=0
REFP 3 C00013 BC00013
CALL JOB:SEARCH-R1
SET P0101 P0006
SFTON P0101
MOVL C00014 BC00014 V=333.3 PL=0
SFTOF
'W9P
MOVL C00015 BC00015 V=666.7
MOVL C00016 BC00016 V=166.7
REFP 3 C00017 BC00017
CALL JOB:SEARCH-R1
SET P0102 P0006
SFTON P0102
MOVL C00018 BC00018 V=166.7 PL=0
REFP 3 C00019 BC00019
CALL JOB:SEARCH-R1
SET P0102 P0006
SFTON P0102
MOVL C00020 BC00020 V=333.3 PL=0
'W9L
MOVL C00021 BC00021 V=666.7
MOVL C00022 BC00022 V=166.7
REFP 3 C00023 BC00023
CALL JOB:SEARCH-R1
SET P0103 P0006
SFTON P0103
MOVL C00024 BC00024 V=166.7 PL=0
REFP 3 C00025 BC00025
CALL JOB:SEARCH-R1
SET P0103 P0006
SFTON P0103
MOVL C00026 BC00026 V=333.3 PL=0
'PRZEJAZ NAD BELKA
MOVL C00027 BC00027 V=666.7
MOVJ C00028 BC00028 VJ=40.00
MOVJ C00029 BC00029 VJ=40.00
MOVJ C00030 BC00030 VJ=40.00
'W1P
MOVJ C00031 BC00031 VJ=20.00 PL=0
MOVL C00032 BC00032 V=166.7 PL=0
REFP 3 C00033 BC00033
CALL JOB:SEARCH-R1
SET P0104 P0006
SFTON P0104
MOVL C00034 BC00034 V=166.7 PL=0
REFP 3 C00035 BC00035
CALL JOB:SEARCH-R1
SET P0104 P0006
SFTON P0104
MOVL C00036 BC00036 V=333.3 PL=0
SFTOF
'W1L
MOVL C00037 BC00037 V=666.7
MOVL C00038 BC00038 V=166.7 PL=0
REFP 3 C00039 BC00039
CALL JOB:SEARCH-R1
SET P0105 P0006
SFTON P0105
MOVL C00040 BC00040 V=166.7 PL=0
REFP 3 C00041 BC00041
CALL JOB:SEARCH-R1
SET P0105 P0006
SFTON P0105
MOVL C00042 BC00042 V=333.3 PL=0
SFTOF
MOVL C00043 BC00043 V=666.7
'W10P
MOVL C00044 BC00044 V=166.7 PL=0
REFP 3 C00045 BC00045
CALL JOB:SEARCH-R1
SET P0106 P0006
SFTON P0106
MOVL C00046 BC00046 V=166.7 PL=0
REFP 3 C00047 BC00047
CALL JOB:SEARCH-R1
SET P0106 P0006
SFTON P0106
MOVL C00048 BC00048 V=333.3 PL=0
SFTOF
'W10L
MOVL C00049 BC00049 V=333.3
MOVL C00050 BC00050 V=166.7 PL=0
REFP 3 C00051 BC00051
CALL JOB:SEARCH-R1
SET P0107 P0006
SFTON P0107
MOVL C00052 BC00052 V=166.7 PL=0
REFP 3 C00053 BC00053
CALL JOB:SEARCH-R1
SET P0107 P0006
SFTON P0107
MOVL C00054 BC00054 V=333.3 PL=0
SFTOF
MOVL C00055 BC00055 V=333.3
'PRZEJAZD
MOVJ C00056 BC00056 VJ=50.00
MOVJ C00057 BC00057 VJ=50.00
MOVJ C00058 BC00058 VJ=60.00
MOVJ C00059 BC00059 VJ=60.00
MOVJ C00060 BC00060 VJ=60.00
MOVJ C00061 BC00061 VJ=60.00 PL=0
MOVL C00062 BC00062 V=166.7 PL=0
REFP 3 C00063 BC00063
CALL JOB:SEARCH-R1
SET P0108 P0006
SFTON P0108
MOVL C00064 BC00064 V=166.7 PL=0
REFP 3 C00065 BC00065
CALL JOB:SEARCH-R1
SET P0108 P0006
SFTON P0108
MOVL C00066 BC00066 V=333.3 PL=0
SFTOF
'W2P
'W2L
MOVL C00067 BC00067 V=666.7
MOVL C00068 BC00068 V=166.7 PL=0
REFP 3 C00069 BC00069
CALL JOB:SEARCH-R1
SET P0109 P0006
SFTON P0109
MOVL C00070 BC00070 V=166.7 PL=0
REFP 3 C00071 BC00071
CALL JOB:SEARCH-R1
SET P0109 P0006
SFTON P0109
MOVL C00072 BC00072 V=333.3 PL=0
SFTOF
MOVJ C00073 BC00073 VJ=25.00
MOVJ C00074 BC00074 VJ=50.00
'W5L
MOVJ C00075 BC00075 VJ=30.00 PL=0
MOVL C00076 BC00076 V=166.7
REFP 3 C00077 BC00077
CALL JOB:SEARCH-R1
SET P0021 P0006
SFTON P0021
MOVL C00078 BC00078 V=166.7
REFP 3 C00079 BC00079
CALL JOB:SEARCH-R1
SET P0021 P0006
SFTON P0021
SFTOF
MOVL C00080 BC00080 V=166.7
'W6L
MOVJ C00081 BC00081 VJ=20.00 PL=0
MOVL C00082 BC00082 V=166.7
REFP 3 C00083 BC00083
CALL JOB:SEARCH-R1
SET P0022 P0006
SFTON P0022
MOVL C00084 BC00084 V=166.7
REFP 3 C00085 BC00085
CALL JOB:SEARCH-R1
SET P0022 P0006
SFTON P0022
SFTOF
MOVL C00086 BC00086 V=166.7
'W6P
MOVL C00087 BC00087 V=333.3 PL=0
REFP 3 C00088 BC00088
CALL JOB:SEARCH-R1
SET P0023 P0006
SFTON P0023
MOVL C00089 BC00089 V=166.7
REFP 3 C00090 BC00090
CALL JOB:SEARCH-R1
SET P0023 P0006
SFTON P0023
SFTOF
MOVL C00091 BC00091 V=166.7
'W5P
MOVJ C00092 BC00092 VJ=20.00 PL=0
MOVL C00093 BC00093 V=166.7
REFP 3 C00094 BC00094
CALL JOB:SEARCH-R1
SET P0024 P0006
SFTON P0024
MOVL C00095 BC00095 V=166.7
REFP 3 C00096 BC00096
CALL JOB:SEARCH-R1
SET P0024 P0006
SFTON P0024
SFTOF
MOVL C00097 BC00097 V=166.7
'W7A
MOVJ C00098 BC00098 VJ=40.00
MOVJ C00099 BC00099 VJ=40.00
MOVJ C00100 BC00100 VJ=40.00
MOVJ C00101 BC00101 VJ=40.00
MOVJ C00102 BC00102 VJ=40.00
MOVJ C00103 BC00103 VJ=40.00
MOVJ C00104 BC00104 VJ=40.00
MOVJ C00105 BC00105 VJ=40.00
MOVL C00106 BC00106 V=250.0
REFP 3 C00107 BC00107
CALL JOB:SEARCH-R1
SET P0280 P0006
SFTON P0280
MOVL C00108 BC00108 V=166.7
MOVL C00109 BC00109 V=250.0
MOVL C00110 BC00110 V=166.7
REFP 3 C00111 BC00111
CALL JOB:SEARCH-R1
SET P0280 P0006
MOVL C00112 BC00112 V=166.7
SFTOF
MOVL C00113 BC00113 V=333.3
MOVL C00114 BC00114 V=166.7
REFP 3 C00115 BC00115
CALL JOB:SEARCH-R1
SET P0290 P0006
SFTON P0290
MOVL C00116 BC00116 V=166.7
REFP 3 C00117 BC00117
CALL JOB:SEARCH-R1
SET P0290 P0006
MOVL C00118 BC00118 V=166.7
MOVJ C00119 BC00119 VJ=20.00
SFTOF
MOVJ C00120 BC00120 VJ=30.00
MOVJ C00121 BC00121 VJ=40.00
MOVJ C00122 BC00122 VJ=40.00
MOVJ C00123 BC00123 VJ=40.00
MOVJ C00124 BC00124 VJ=40.00
MOVJ C00125 BC00125 VJ=50.00
'W7B
MOVJ C00126 BC00126 VJ=50.00
MOVJ C00127 BC00127 VJ=50.00
MOVJ C00128 BC00128 VJ=30.00
MOVJ C00129 BC00129 VJ=20.00
MOVL C00130 BC00130 V=166.7
REFP 3 C00131 BC00131
CALL JOB:SEARCH-R1
SET P0281 P0006
MOVL C00132 BC00132 V=166.7
SFTON P0281
MOVL C00133 BC00133 V=166.7
MOVL C00134 BC00134 V=166.7
REFP 3 C00135 BC00135
CALL JOB:SEARCH-R1
SET P0281 P0006
MOVJ C00136 BC00136 VJ=15.00
SFTOF
MOVJ C00137 BC00137 VJ=20.00
MOVL C00138 BC00138 V=166.7
REFP 3 C00139 BC00139
CALL JOB:SEARCH-R1
SET P0291 P0006
MOVL C00140 BC00140 V=166.7
MOVL C00141 BC00141 V=166.7
REFP 3 C00142 BC00142
CALL JOB:SEARCH-R1
SET P0291 P0006
MOVL C00143 BC00143 V=166.7
COMM MOVJ C00144 BC00144 VJ=40.00
COMM MOVJ C00145 BC00145 VJ=50.00
COMM 'W5L
COMM MOVJ C00146 BC00146 VJ=30.00 PL=0
COMM SET I020 110
COMM CALL JOB:SEARCH_Z-40_Z1_X40
COMM MOVL C00147 BC00147 V=166.7
COMM 'W6L
COMM MOVJ C00148 BC00148 VJ=20.00 PL=0
COMM SET I020 112
COMM CALL JOB:SEARCH_Z-40_Z1_X40
COMM MOVL C00149 BC00149 V=166.7
COMM 'W6P
COMM MOVL C00150 BC00150 V=150.0 PL=0
COMM SET I020 113
COMM CALL JOB:SEARCH_Z-40_Z1_X40
COMM MOVL C00151 BC00151 V=166.7
COMM 'W5P
COMM MOVJ C00152 BC00152 VJ=20.00 PL=0
COMM SET I020 111
COMM CALL JOB:SEARCH_Z-40_Z1_X40
COMM MOVL C00153 BC00153 V=166.7
COMM 'W7A
COMM MOVJ C00154 BC00154 VJ=40.00
COMM MOVJ C00155 BC00155 VJ=40.00
COMM MOVJ C00156 BC00156 VJ=40.00
COMM MOVJ C00157 BC00157 VJ=40.00
COMM MOVJ C00158 BC00158 VJ=40.00
COMM MOVJ C00159 BC00159 VJ=40.00
COMM MOVJ C00160 BC00160 VJ=40.00
COMM MOVJ C00161 BC00161 VJ=40.00
COMM MOVL C00162 BC00162 V=250.0
COMM REFP 3 C00163 BC00163
COMM CALL JOB:SEARCH-R1
COMM SET P0280 P0006
COMM SFTON P0280
COMM MOVL C00164 BC00164 V=166.7
COMM MOVL C00165 BC00165 V=250.0
COMM MOVL C00166 BC00166 V=166.7
COMM REFP 3 C00167 BC00167
COMM CALL JOB:SEARCH-R1
COMM SET P0280 P0006
COMM MOVL C00168 BC00168 V=166.7
COMM SFTOF
COMM MOVL C00169 BC00169 V=333.3
COMM MOVL C00170 BC00170 V=166.7
COMM REFP 3 C00171 BC00171
COMM CALL JOB:SEARCH-R1
COMM SET P0290 P0006
COMM SFTON P0290
COMM MOVL C00172 BC00172 V=166.7
COMM REFP 3 C00173 BC00173
COMM CALL JOB:SEARCH-R1
COMM SET P0290 P0006
COMM MOVL C00174 BC00174 V=166.7
COMM 'DOKONCZYC SEARCH
COMM 'DOKONCZYC SEARCH
COMM MOVJ C00175 BC00175 VJ=20.00
COMM SFTOF
COMM MOVJ C00176 BC00176 VJ=30.00
COMM MOVJ C00177 BC00177 VJ=40.00
COMM MOVJ C00178 BC00178 VJ=40.00
COMM MOVJ C00179 BC00179 VJ=40.00
COMM MOVJ C00180 BC00180 VJ=40.00
COMM MOVJ C00181 BC00181 VJ=50.00
COMM 'W7B
COMM MOVJ C00182 BC00182 VJ=50.00
COMM MOVJ C00183 BC00183 VJ=50.00
COMM MOVJ C00184 BC00184 VJ=30.00
COMM MOVJ C00185 BC00185 VJ=20.00
COMM MOVL C00186 BC00186 V=166.7
COMM REFP 3 C00187 BC00187
COMM CALL JOB:SEARCH-R1
COMM SET P0281 P0006
COMM MOVL C00188 BC00188 V=166.7
COMM SFTON P0281
COMM MOVL C00189 BC00189 V=166.7
COMM MOVL C00190 BC00190 V=166.7
COMM REFP 3 C00191 BC00191
COMM CALL JOB:SEARCH-R1
COMM SET P0281 P0006
COMM MOVJ C00192 BC00192 VJ=15.00
COMM SFTOF
COMM MOVJ C00193 BC00193 VJ=20.00
COMM MOVL C00194 BC00194 V=166.7
COMM REFP 3 C00195 BC00195
COMM CALL JOB:SEARCH-R1
COMM SET P0291 P0006
COMM MOVL C00196 BC00196 V=166.7
COMM MOVL C00197 BC00197 V=166.7
COMM REFP 3 C00198 BC00198
COMM CALL JOB:SEARCH-R1
COMM SET P0291 P0006
COMM MOVL C00199 BC00199 V=166.7
COMM 'DOKONCZYC SEARCH
COMM 'DOKONCZYC SEARCH
COMM 'DOKONCZYC SEARCH
MOVJ C00200 BC00200 VJ=30.00
MOVJ C00201 BC00201 VJ=30.00
MOVJ C00202 BC00202 VJ=50.00
MOVJ C00203 BC00203 VJ=50.00
'------------------------
'------------------------
'PRAWA STRONA PROFIL GORA
'------------------------
'------------------------
MOVJ C00204 BC00204 VJ=50.00
MOVJ C00205 BC00205 VJ=50.00
MOVJ C00206 BC00206 VJ=50.00
MOVJ C00207 BC00207 VJ=20.00
MOVJ C00208 BC00208 VJ=50.00
'------------------------
'W14A L
'------------------------
SFTOF
MOVJ C00209 BC00209 VJ=50.00
MOVJ C00210 BC00210 VJ=30.00
MOVL C00211 BC00211 V=166.7 PL=0
REFP 3 C00212 BC00212
CALL JOB:SEARCH-R1
SET P0300 P0006
SFTON P0300
MOVL C00213 BC00213 V=166.7 PL=0
REFP 3 C00214 BC00214
CALL JOB:SEARCH-R1
SET P0300 P0006
SFTON P0300
MOVL C00215 BC00215 V=166.7 PL=0
SFTOF
'------------------------
'W14A P
'------------------------
SFTOF
MOVJ C00216 BC00216 VJ=50.00
MOVJ C00217 BC00217 VJ=50.00
MOVL C00218 BC00218 V=166.7 PL=0
REFP 3 C00219 BC00219
CALL JOB:SEARCH-R1
SET P0301 P0006
SFTON P0301
MOVL C00220 BC00220 V=166.7 PL=0
REFP 3 C00221 BC00221
CALL JOB:SEARCH-R1
SET P0301 P0006
SFTON P0301
MOVL C00222 BC00222 V=166.7 PL=0
SFTOF
'------------------------
'W19A L
'------------------------
SFTOF
MOVJ C00223 BC00223 VJ=50.00
MOVL C00224 BC00224 V=200.0 PL=0
REFP 3 C00225 BC00225
CALL JOB:SEARCH-R1
SET P0302 P0006
SFTON P0302
MOVL C00226 BC00226 V=166.7 PL=0
REFP 3 C00227 BC00227
CALL JOB:SEARCH-R1
SET P0302 P0006
SFTON P0302
MOVL C00228 BC00228 V=250.0 PL=0
SFTOF
'------------------------
'W19A P
'------------------------
SFTOF
MOVJ C00229 BC00229 VJ=50.00
MOVL C00230 BC00230 V=166.7 PL=0
REFP 3 C00231 BC00231
CALL JOB:SEARCH-R1
SET P0303 P0006
SFTON P0303
MOVL C00232 BC00232 V=166.7 PL=0
REFP 3 C00233 BC00233
CALL JOB:SEARCH-R1
SET P0303 P0006
SFTON P0303
MOVL C00234 BC00234 V=166.7 PL=0
SFTOF
'------------------------
'W13A L
'------------------------
SFTOF
MOVJ C00235 BC00235 VJ=50.00
MOVL C00236 BC00236 V=166.7 PL=0
REFP 3 C00237 BC00237
CALL JOB:SEARCH-R1
SET P0304 P0006
SFTON P0304
MOVL C00238 BC00238 V=166.7 PL=0
REFP 3 C00239 BC00239
CALL JOB:SEARCH-R1
SET P0304 P0006
SFTON P0304
MOVL C00240 BC00240 V=166.7 PL=0
SFTOF
'------------------------
'W13A P
'------------------------
SFTOF
MOVJ C00241 BC00241 VJ=50.00
MOVL C00242 BC00242 V=200.0 PL=0
REFP 3 C00243 BC00243
CALL JOB:SEARCH-R1
SET P0305 P0006
SFTON P0305
MOVL C00244 BC00244 V=166.7 PL=0
REFP 3 C00245 BC00245
CALL JOB:SEARCH-R1
SET P0305 P0006
SFTON P0305
MOVL C00246 BC00246 V=250.0 PL=0
SFTOF
'------------------------
'W18A L
'------------------------
SFTOF
MOVJ C00247 BC00247 VJ=50.00
MOVL C00248 BC00248 V=200.0 PL=0
REFP 3 C00249 BC00249
CALL JOB:SEARCH-R1
SET P0306 P0006
SFTON P0306
MOVL C00250 BC00250 V=166.7 PL=0
REFP 3 C00251 BC00251
CALL JOB:SEARCH-R1
SET P0306 P0006
SFTON P0306
MOVL C00252 BC00252 V=166.7 PL=0
SFTOF
'------------------------
'W18A P
'------------------------
SFTOF
MOVJ C00253 BC00253 VJ=50.00
MOVL C00254 BC00254 V=200.0 PL=0
REFP 3 C00255 BC00255
CALL JOB:SEARCH-R1
SET P0307 P0006
SFTON P0307
MOVL C00256 BC00256 V=166.7 PL=0
REFP 3 C00257 BC00257
CALL JOB:SEARCH-R1
SET P0307 P0006
SFTON P0307
MOVL C00258 BC00258 V=166.7 PL=0
SFTOF
'------------------------
'W15A L
'------------------------
SFTOF
MOVJ C00259 BC00259 VJ=50.00
MOVL C00260 BC00260 V=200.0 PL=0
REFP 3 C00261 BC00261
CALL JOB:SEARCH-R1
SET P0308 P0006
SFTON P0308
MOVL C00262 BC00262 V=166.7 PL=0
REFP 3 C00263 BC00263
CALL JOB:SEARCH-R1
SET P0308 P0006
SFTON P0308
MOVL C00264 BC00264 V=166.7 PL=0
SFTOF
'------------------------
'W15A P
'------------------------
SFTOF
MOVJ C00265 BC00265 VJ=50.00
MOVL C00266 BC00266 V=166.7 PL=0
REFP 3 C00267 BC00267
CALL JOB:SEARCH-R1
SET P0309 P0006
SFTON P0309
MOVL C00268 BC00268 V=166.7 PL=0
REFP 3 C00269 BC00269
CALL JOB:SEARCH-R1
SET P0309 P0006
SFTON P0309
MOVL C00270 BC00270 V=166.7 PL=0
SFTOF
MOVL C00271 BC00271 V=333.3
'------------------------
'W17A L
'------------------------
MOVL C00272 BC00272 V=500.0
SFTOF
MOVJ C00273 BC00273 VJ=20.00
MOVL C00274 BC00274 V=166.7 PL=0
REFP 3 C00275 BC00275
CALL JOB:SEARCH-R1
SET P0310 P0006
SFTON P0310
MOVL C00276 BC00276 V=166.7 PL=0
REFP 3 C00277 BC00277
CALL JOB:SEARCH-R1
SET P0310 P0006
SFTON P0310
MOVL C00278 BC00278 V=166.7 PL=0
SFTOF
'------------------------
'W17A P
'------------------------
SFTOF
MOVL C00279 BC00279 V=416.7
MOVL C00280 BC00280 V=166.7 PL=0
REFP 3 C00281 BC00281
CALL JOB:SEARCH-R1
SET P0311 P0006
SFTON P0311
MOVL C00282 BC00282 V=166.7 PL=0
REFP 3 C00283 BC00283
CALL JOB:SEARCH-R1
SET P0311 P0006
SFTON P0311
MOVL C00284 BC00284 V=166.7 PL=0
SFTOF
MOVJ C00285 BC00285 VJ=10.00
MOVJ C00286 BC00286 VJ=20.00
MOVJ C00287 BC00287 VJ=50.00
MOVJ C00288 BC00288 VJ=50.00
MOVJ C00289 BC00289 VJ=70.00
MOVJ C00290 BC00290 VJ=30.00
MOVJ C00291 BC00291 VJ=30.00
'------------------------
'------------------------
'LEWA STRONA PROFIL GORA
'------------------------
'------------------------
MOVJ C00292 BC00292 VJ=30.00
MOVJ C00293 BC00293 VJ=30.00
MOVJ C00294 BC00294 VJ=30.00
'------------------------
'W17B L
'------------------------
SFTOF
MOVJ C00295 BC00295 VJ=15.00
MOVL C00296 BC00296 V=166.7 PL=0
REFP 3 C00297 BC00297
CALL JOB:SEARCH-R1
SET P0350 P0006
SFTON P0350
MOVL C00298 BC00298 V=166.7 PL=0
REFP 3 C00299 BC00299
CALL JOB:SEARCH-R1
SET P0350 P0006
SFTON P0350
MOVL C00300 BC00300 V=166.7 PL=0
SFTOF
'------------------------
'W17B P
'------------------------
SFTOF
MOVL C00301 BC00301 V=333.3
MOVL C00302 BC00302 V=166.7 PL=0
REFP 3 C00303 BC00303
CALL JOB:SEARCH-R1
SET P0351 P0006
SFTON P0351
MOVL C00304 BC00304 V=166.7 PL=0
REFP 3 C00305 BC00305
CALL JOB:SEARCH-R1
SET P0351 P0006
SFTON P0351
MOVL C00306 BC00306 V=166.7 PL=0
SFTOF
'POPRAWID DOJAZD
'------------------------
'W15B L
'------------------------
SFTOF
MOVJ C00307 BC00307 VJ=10.00
MOVL C00308 BC00308 V=166.7 PL=0
REFP 3 C00309 BC00309
CALL JOB:SEARCH-R1
SET P0352 P0006
SFTON P0352
MOVL C00310 BC00310 V=166.7 PL=0
REFP 3 C00311 BC00311
CALL JOB:SEARCH-R1
SET P0352 P0006
SFTON P0352
MOVL C00312 BC00312 V=166.7 PL=0
SFTOF
'------------------------
'W15B P
'------------------------
SFTOF
MOVJ C00313 BC00313 VJ=20.00
MOVL C00314 BC00314 V=166.7 PL=0
REFP 3 C00315 BC00315
CALL JOB:SEARCH-R1
SET P0353 P0006
SFTON P0353
MOVL C00316 BC00316 V=166.7 PL=0
REFP 3 C00317 BC00317
CALL JOB:SEARCH-R1
SET P0353 P0006
SFTON P0353
MOVL C00318 BC00318 V=166.7 PL=0
SFTOF
'------------------------
'W18B L
'------------------------
SFTOF
MOVJ C00319 BC00319 VJ=50.00
MOVL C00320 BC00320 V=166.7 PL=0
REFP 3 C00321 BC00321
CALL JOB:SEARCH-R1
SET P0354 P0006
SFTON P0354
MOVL C00322 BC00322 V=166.7 PL=0
REFP 3 C00323 BC00323
CALL JOB:SEARCH-R1
SET P0354 P0006
SFTON P0354
MOVL C00324 BC00324 V=166.7 PL=0
SFTOF
'------------------------
'W18B P
'------------------------
SFTOF
MOVJ C00325 BC00325 VJ=50.00
MOVL C00326 BC00326 V=166.7 PL=0
REFP 3 C00327 BC00327
CALL JOB:SEARCH-R1
SET P0355 P0006
SFTON P0355
MOVL C00328 BC00328 V=166.7 PL=0
REFP 3 C00329 BC00329
CALL JOB:SEARCH-R1
SET P0355 P0006
SFTON P0355
MOVL C00330 BC00330 V=166.7 PL=0
SFTOF
'------------------------
'W13B L
'------------------------
SFTOF
MOVJ C00331 BC00331 VJ=50.00
MOVL C00332 BC00332 V=166.7 PL=0
REFP 3 C00333 BC00333
CALL JOB:SEARCH-R1
SET P0356 P0006
SFTON P0356
MOVL C00334 BC00334 V=166.7 PL=0
REFP 3 C00335 BC00335
CALL JOB:SEARCH-R1
SET P0356 P0006
SFTON P0356
MOVL C00336 BC00336 V=166.7 PL=0
SFTOF
'------------------------
'W13B P
'------------------------
SFTOF
MOVJ C00337 BC00337 VJ=50.00
MOVL C00338 BC00338 V=166.7 PL=0
REFP 3 C00339 BC00339
CALL JOB:SEARCH-R1
SET P0357 P0006
SFTON P0357
MOVL C00340 BC00340 V=166.7 PL=0
REFP 3 C00341 BC00341
CALL JOB:SEARCH-R1
SET P0357 P0006
SFTON P0357
MOVL C00342 BC00342 V=166.7 PL=0
SFTOF
'------------------------
'W19B L
'------------------------
SFTOF
MOVJ C00343 BC00343 VJ=50.00
MOVL C00344 BC00344 V=166.7 PL=0
REFP 3 C00345 BC00345
CALL JOB:SEARCH-R1
SET P0358 P0006
SFTON P0358
MOVL C00346 BC00346 V=166.7 PL=0
REFP 3 C00347 BC00347
CALL JOB:SEARCH-R1
SET P0358 P0006
SFTON P0358
MOVL C00348 BC00348 V=166.7 PL=0
SFTOF
'------------------------
'W19B P
'------------------------
SFTOF
MOVJ C00349 BC00349 VJ=50.00
MOVL C00350 BC00350 V=166.7 PL=0
REFP 3 C00351 BC00351
CALL JOB:SEARCH-R1
SET P0359 P0006
SFTON P0359
MOVL C00352 BC00352 V=166.7 PL=0
REFP 3 C00353 BC00353
CALL JOB:SEARCH-R1
SET P0359 P0006
SFTON P0359
MOVL C00354 BC00354 V=166.7 PL=0
SFTOF
'------------------------
'W14B L
'------------------------
SFTOF
MOVJ C00355 BC00355 VJ=50.00
MOVL C00356 BC00356 V=166.7 PL=0
REFP 3 C00357 BC00357
CALL JOB:SEARCH-R1
SET P0360 P0006
SFTON P0360
MOVL C00358 BC00358 V=166.7 PL=0
REFP 3 C00359 BC00359
CALL JOB:SEARCH-R1
SET P0360 P0006
SFTON P0360
MOVL C00360 BC00360 V=166.7 PL=0
SFTOF
'------------------------
'W14B P
'------------------------
SFTOF
MOVJ C00361 BC00361 VJ=50.00
MOVL C00362 BC00362 V=166.7 PL=0
REFP 3 C00363 BC00363
CALL JOB:SEARCH-R1
SET P0361 P0006
SFTON P0361
MOVL C00364 BC00364 V=166.7 PL=0
REFP 3 C00365 BC00365
CALL JOB:SEARCH-R1
SET P0361 P0006
SFTON P0361
MOVL C00366 BC00366 V=166.7 PL=0
SFTOF
MOVJ C00367 BC00367 VJ=50.00
MOVJ C00368 BC00368 VJ=50.00
MOVJ C00369 BC00369 VJ=50.00
MOVJ C00370 BC00370 VJ=50.00
'WELD
'WELD
'WELD
MOVJ C00371 BC00371 VJ=10.00
'**********************
'**********************
'POCZATEK SPAWANIA DOL
'**********************
'**********************
''
'**********************
'W1
'**********************
MOVJ C00372 BC00372 VJ=50.00
MOVJ C00373 BC00373 VJ=40.00
MOVL C00374 BC00374 V=166.7
SFTON P0104
MOVL C00375 BC00375 V=166.7
MACRO1 MJ#(0) ARGF24
ARCON
SFTON P0105
MOVL C00376 BC00376 V=11.7
ARCOF
SFTOF
MOVJ C00377 BC00377 VJ=20.00
MOVJ C00378 BC00378 VJ=30.00
MOVJ C00379 BC00379 VJ=50.00
MOVJ C00380 BC00380 VJ=40.00
MOVJ C00381 BC00381 VJ=20.00
'**********************
'W2
'**********************
SFTON P0108
MOVL C00382 BC00382 V=166.7
ARCON
SFTON P0109
MOVL C00383 BC00383 V=11.7
MOVL C00384 BC00384 V=11.7
ARCOF
SFTOF
MOVL C00385 BC00385 V=333.3
MOVJ C00386 BC00386 VJ=40.00
MOVJ C00387 BC00387 VJ=70.00
MOVJ C00388 BC00388 VJ=20.00
MOVL C00389 BC00389 V=666.7
'**********************
'W3
'**********************
SFTON P0101
MOVL C00390 BC00390 V=166.7
ARCON
SFTON P0100
MOVL C00391 BC00391 V=11.7
ARCOF
MOVL C00392 BC00392 V=166.7
SFTOF
MOVJ C00393 BC00393 VJ=30.00
MOVJ C00394 BC00394 VJ=30.00
MOVJ C00395 BC00395 VJ=50.00
MOVJ C00396 BC00396 VJ=30.00
MOVJ C00397 BC00397 VJ=40.00
'**********************
'W5
'**********************
MOVJ C00398 BC00398 VJ=50.00
MOVJ C00399 BC00399 VJ=25.00
MOVJ C00400 BC00400 VJ=30.00
MOVL C00401 BC00401 V=333.3
'**********************
MACRO1 MJ#(0) ARGF9
SFTON P0024
MOVL C00402 BC00402 V=166.7
ARCON
SFTON P0021
MOVL C00403 BC00403 V=10.8
ARCOF
SFTOF
MOVJ C00404 BC00404 VJ=20.00
MOVJ C00405 BC00405 VJ=20.00
'**********************
'W6
'**********************
MACRO1 MJ#(0) ARGF9
SFTON P0023
MOVL C00406 BC00406 V=250.0
ARCON
SFTON P0022
MOVL C00407 BC00407 V=10.8
ARCOF
SFTOF
MOVJ C00408 BC00408 VJ=10.00
MOVJ C00409 BC00409 VJ=30.00
MOVJ C00410 BC00410 VJ=40.00
MOVJ C00411 BC00411 VJ=40.00
MOVJ C00412 BC00412 VJ=40.00
MOVJ C00413 BC00413 VJ=40.00
MOVJ C00414 BC00414 VJ=20.00
MOVJ C00415 BC00415 VJ=10.00
MOVJ C00416 BC00416 VJ=20.00
MOVL C00417 BC00417 V=166.7
MACRO1 MJ#(0) ARGF14
MOVL C00418 BC00418 V=166.7
SFTON P0280
MOVL C00419 BC00419 V=166.7 PL=0
ARCON ASF#(22)
MOVL C00420 BC00420 V=9.2
MOVL C00421 BC00421 V=9.2
SFTON P0290
MOVL C00422 BC00422 V=9.2
MOVL C00423 BC00423 V=9.2
ARCOF
SFTOF
MOVL C00424 BC00424 V=250.0
MOVL C00425 BC00425 V=416.7
MOVJ C00426 BC00426 VJ=30.00
MOVJ C00427 BC00427 VJ=30.00
MOVJ C00428 BC00428 VJ=30.00
MOVJ C00429 BC00429 VJ=30.00
MOVJ C00430 BC00430 VJ=30.00
'7b
MOVL C00431 BC00431 V=333.3
MOVL C00432 BC00432 V=333.3
SFTON P0281
MOVL C00433 BC00433 V=166.7 PL=0
ARCON ASF#(22)
MOVL C00434 BC00434 V=9.2
MOVL C00435 BC00435 V=9.2
SFTON P0291
MOVL C00436 BC00436 V=9.2
MOVL C00437 BC00437 V=9.2
MOVL C00438 BC00438 V=9.2
ARCOF
SFTOF
'TUTAJ DODAC 7
'TUTAJ DODAC 7
'TUTAJ DODAC 7
MOVL C00439 BC00439 V=333.3
MOVL C00440 BC00440 V=333.3
MOVL C00441 BC00441 V=333.3
COMM '**********************
COMM 'W5
COMM '**********************
COMM MACRO1 MJ#(0) ARGF9
COMM SFTON P0021
COMM MOVL P0111 BP111 V=66.7
COMM ARCON
COMM MOVL P0110 BP110 V=10.0
COMM ARCOF
COMM SFTOF
COMM MOVJ C00442 BC00442 VJ=20.00
COMM MOVJ C00443 BC00443 VJ=20.00
COMM '**********************
COMM 'W6
COMM '**********************
COMM MACRO1 MJ#(0) ARGF9
COMM SFTON P0023
COMM MOVL P0113 BP113 V=66.7
COMM ARCON
COMM MOVL P0112 BP112 V=10.8
COMM ARCOF
COMM SFTOF
COMM MOVJ C00444 BC00444 VJ=10.00
COMM MOVJ C00445 BC00445 VJ=30.00
COMM MOVJ C00446 BC00446 VJ=30.00
COMM MOVJ C00447 BC00447 VJ=40.00
COMM MOVJ C00448 BC00448 VJ=40.00
COMM MOVJ C00449 BC00449 VJ=40.00
COMM MOVJ C00450 BC00450 VJ=40.00
COMM MOVJ C00451 BC00451 VJ=20.00
COMM MOVJ C00452 BC00452 VJ=10.00
COMM MOVJ C00453 BC00453 VJ=20.00
COMM MOVL C00454 BC00454 V=166.7
COMM MACRO1 MJ#(0) ARGF14
COMM MOVL C00455 BC00455 V=166.7
COMM SFTON P0280
COMM MOVL C00456 BC00456 V=166.7 PL=0
COMM ARCON ASF#(22)
COMM MOVL C00457 BC00457 V=9.2
COMM MOVL C00458 BC00458 V=9.2
COMM SFTON P0281
COMM MOVL C00459 BC00459 V=9.2
COMM MOVL C00460 BC00460 V=9.2
COMM ARCOF
COMM SFTOF
COMM MOVL C00461 BC00461 V=250.0
COMM MOVL C00462 BC00462 V=416.7
COMM MOVJ C00463 BC00463 VJ=30.00
COMM MOVJ C00464 BC00464 VJ=30.00
COMM MOVJ C00465 BC00465 VJ=30.00
COMM MOVJ C00466 BC00466 VJ=30.00
COMM MOVJ C00467 BC00467 VJ=30.00
COMM '7b
COMM MOVL C00468 BC00468 V=333.3
COMM MOVL C00469 BC00469 V=333.3
COMM SFTON P0281
COMM MOVL C00470 BC00470 V=166.7 PL=0
COMM ARCON ASF#(22)
COMM MOVL C00471 BC00471 V=9.2
COMM MOVL C00472 BC00472 V=9.2
COMM SFTON P0291
COMM MOVL C00473 BC00473 V=9.2
COMM MOVL C00474 BC00474 V=9.2
COMM MOVL C00475 BC00475 V=9.2
COMM ARCOF
COMM SFTOF
COMM 'TUTAJ DODAC 7
COMM 'TUTAJ DODAC 7
COMM 'TUTAJ DODAC 7
COMM MOVL C00476 BC00476 V=333.3
COMM MOVL C00477 BC00477 V=333.3
COMM MOVL C00478 BC00478 V=333.3
MOVJ C00479 BC00479 VJ=20.00
MOVJ C00480 BC00480 VJ=30.00
MOVJ C00481 BC00481 VJ=50.00
MOVJ C00482 BC00482 VJ=50.00
MOVJ C00483 BC00483 VJ=40.00
MOVJ C00484 BC00484 VJ=10.00
'**********************
'W9
'**********************
SFTON P0103
MACRO1 MJ#(0) ARGF24
MOVL C00485 BC00485 V=166.7
ARCON
SFTON P0102
MOVL C00486 BC00486 V=11.7
ARCOF
SFTOF
MOVL C00487 BC00487 V=166.7
MOVJ C00488 BC00488 VJ=40.00
MOVJ C00489 BC00489 VJ=70.00
MOVJ C00490 BC00490 VJ=50.00
MOVJ C00491 BC00491 VJ=20.00
'**********************
'W10
'**********************
MOVL C00492 BC00492 V=333.3
SFTON P0106
MOVL C00493 BC00493 V=166.7
ARCON
SFTON P0107
MOVL C00494 BC00494 V=11.7
ARCOF
SFTOF
MOVL C00495 BC00495 V=333.3
MOVJ C00496 BC00496 VJ=50.00
'**********************
'**********************
'POCZATEK SPAWANIA BOKI
'**********************
'**********************
MOVJ C00497 BC00497 VJ=50.00
MOVJ C00498 BC00498 VJ=50.00
'**********************
'W13A
'**********************
SFTON P0305
MOVL C00499 BC00499 V=250.0 PL=0
SFTOF
MACRO1 MJ#(0) ARGF10
ARCON
SFTON P0304
MOVL C00500 BC00500 V=10.8
ARCOF
SFTOF
MOVL C00501 BC00501 V=250.0
'W13B
MOVJ C00502 BC00502 VJ=30.00
MOVJ C00503 BC00503 VJ=50.00
MOVL C00504 BC00504 V=500.0
'**********************
'W13B
'**********************
SFTON P0356
MOVL C00505 BC00505 V=133.3 PL=0
SFTOF
ARCON
SFTON P0357
MOVL C00506 BC00506 V=10.8
ARCOF
SFTOF
MOVL C00507 BC00507 V=250.0
MOVJ C00508 BC00508 VJ=30.00
MOVJ C00509 BC00509 VJ=40.00
MOVJ C00510 BC00510 VJ=30.00
MOVJ C00511 BC00511 VJ=30.00
'**********************
'W14A
'**********************
MOVL C00512 BC00512 V=250.0
SFTON P0301
MOVL C00513 BC00513 V=50.0 PL=0
SFTOF
ARCON
SFTON P0300
MOVL C00514 BC00514 V=10.8
MOVL C00515 BC00515 V=10.8
MOVL C00516 BC00516 V=10.8
ARCOF
SFTOF
MOVL C00517 BC00517 V=150.0
MOVJ C00518 BC00518 VJ=40.00
MOVJ C00519 BC00519 VJ=30.00
MOVJ C00520 BC00520 VJ=30.00
MOVJ C00521 BC00521 VJ=30.00
MOVJ C00522 BC00522 VJ=30.00
'**********************
'W14B
'**********************
SFTON P0360
MOVL C00523 BC00523 V=333.3
MOVL C00524 BC00524 V=166.7 PL=0
SFTOF
ARCON
SFTON P0361
MOVL C00525 BC00525 V=10.8
MOVL C00526 BC00526 V=10.8
MOVL C00527 BC00527 V=10.8
ARCOF
SFTOF
MOVL C00528 BC00528 V=250.0
MOVJ C00529 BC00529 VJ=40.00
MOVJ C00530 BC00530 VJ=40.00
MOVJ C00531 BC00531 VJ=30.00
MOVJ C00532 BC00532 VJ=40.00
MOVJ C00533 BC00533 VJ=30.00
MOVJ C00534 BC00534 VJ=30.00
MOVJ C00535 BC00535 VJ=30.00
MOVJ C00536 BC00536 VJ=30.00
MOVJ C00537 BC00537 VJ=30.00
'**********************
'W15A
'**********************
SFTON P0309
MOVL C00538 BC00538 V=166.7
MOVL C00539 BC00539 V=166.7 PL=0
SFTOF
ARCON
SFTON P0308
MOVL C00540 BC00540 V=10.8
ARCOF
SFTOF
MOVL C00541 BC00541 V=150.0
MOVJ C00542 BC00542 VJ=30.00
MOVJ C00543 BC00543 VJ=50.00
MOVJ C00544 BC00544 VJ=50.00
MOVJ C00545 BC00545 VJ=50.00
MOVJ C00546 BC00546 VJ=50.00
MOVJ C00547 BC00547 VJ=50.00
'**********************
'W15B
'**********************
SFTON P0352
MOVL C00548 BC00548 V=250.0
MOVL C00549 BC00549 V=83.3 PL=0
SFTOF
ARCON
SFTON P0353
MOVL C00550 BC00550 V=10.8
ARCOF
MOVL C00551 BC00551 V=66.7
SFTOF
MOVJ C00552 BC00552 VJ=40.00
MOVJ C00553 BC00553 VJ=50.00
MOVJ C00554 BC00554 VJ=50.00
'BRAK W TEJ DLUGOSCI
'**********************
'W16A
'**********************
'**********************
'W16B
'**********************
'BRAK W TEJ DLUGOSCI
'**********************
'W17A
'**********************
MOVJ C00555 BC00555 VJ=50.00
MOVJ C00556 BC00556 VJ=50.00
'**********************
'W17A
'**********************
SFTON P0310
MOVL C00557 BC00557 V=333.3
MOVL C00558 BC00558 V=166.7 PL=0
SFTOF
ARCON
SFTON P0311
MOVL C00559 BC00559 V=10.8
ARCOF
SFTOF
MOVL C00560 BC00560 V=333.3
MOVJ C00561 BC00561 VJ=30.00
MOVJ C00562 BC00562 VJ=30.00
MOVJ C00563 BC00563 VJ=50.00
MOVJ C00564 BC00564 VJ=50.00
MOVJ C00565 BC00565 VJ=50.00
MOVJ C00566 BC00566 VJ=50.00
MOVJ C00567 BC00567 VJ=50.00
MOVJ C00568 BC00568 VJ=30.00
MOVJ C00569 BC00569 VJ=30.00
'**********************
'W17B
'**********************
SFTON P0351
MOVL C00570 BC00570 V=166.7
MOVL C00571 BC00571 V=166.7 PL=0
SFTOF
ARCON
SFTON P0350
MOVL C00572 BC00572 V=10.8
ARCOF
SFTOF
MOVL C00573 BC00573 V=250.0
MOVJ C00574 BC00574 VJ=30.00
MOVJ C00575 BC00575 VJ=30.00
MOVJ C00576 BC00576 VJ=30.00
MOVJ C00577 BC00577 VJ=30.00
MOVJ C00578 BC00578 VJ=40.00
'**********************
'W18A
'**********************
SFTON P0306
MOVL C00579 BC00579 V=333.3
MOVL C00580 BC00580 V=166.7 PL=0
SFTOF
ARCON
SFTON P0307
MOVL C00581 BC00581 V=10.8
ARCOF
SFTOF
MOVL C00582 BC00582 V=250.0
MOVJ C00583 BC00583 VJ=30.00
MOVJ C00584 BC00584 VJ=30.00
MOVJ C00585 BC00585 VJ=50.00
MOVJ C00586 BC00586 VJ=50.00
MOVJ C00587 BC00587 VJ=50.00
'**********************
'W18B
'**********************
SFTON P0355
MOVL C00588 BC00588 V=166.7
MOVL C00589 BC00589 V=166.7 PL=0
SFTOF
ARCON
SFTON P0354
MOVL C00590 BC00590 V=10.8
ARCOF
MOVL C00591 BC00591 V=250.0
SFTOF
MOVJ C00592 BC00592 VJ=30.00
MOVJ C00593 BC00593 VJ=30.00
MOVJ C00594 BC00594 VJ=40.00
MOVJ C00595 BC00595 VJ=50.00
MOVJ C00596 BC00596 VJ=30.00
'**********************
'W19A
'**********************
MOVL C00597 BC00597 V=166.7
SFTON P0303
MOVL C00598 BC00598 V=166.7 PL=0
SFTOF
ARCON
SFTON P0302
MOVL C00599 BC00599 V=10.8
ARCOF
SFTOF
MOVL C00600 BC00600 V=150.0
MOVJ C00601 BC00601 VJ=30.00
MOVJ C00602 BC00602 VJ=50.00
MOVJ C00603 BC00603 VJ=50.00
'**********************
'W19B
'**********************
SFTON P0358
MOVL C00604 BC00604 V=500.0
MOVL C00605 BC00605 V=166.7 PL=0
SFTOF
ARCON
SFTON P0359
MOVL C00606 BC00606 V=10.8
ARCOF
SFTOF
MOVL C00607 BC00607 V=250.0
MOVJ C00608 BC00608 VJ=40.00
MOVJ C00609 BC00609 VJ=50.00
CALL JOB:MOVE_OUT_OF_TUNNEL
END
